Universal Robots URScript: camisa.script

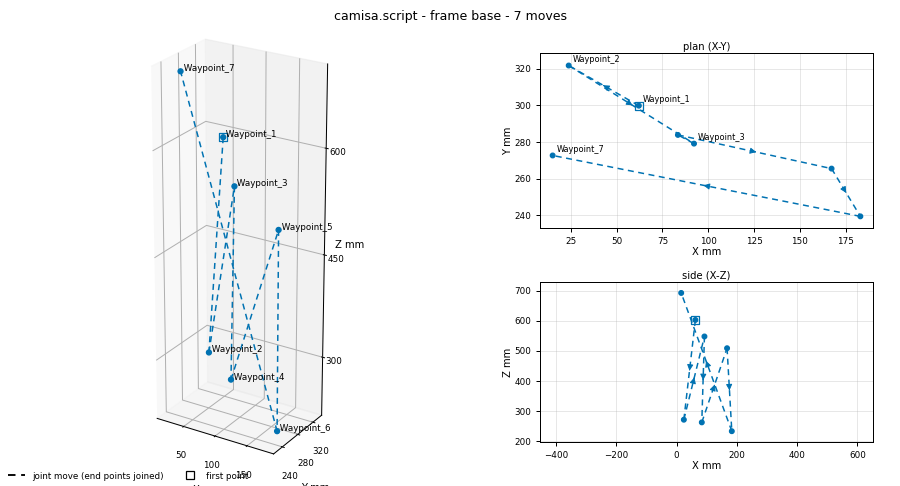
[picture p0: tool path of camisa.script in frame base, 7 of 7 moves have a stored position in this frame; points joined in program order, loops and branches not executed]
def camisa():
  set_tcp(p[0.0,0.0,0.0777,0.0,0.0,0.0])
  set_payload(0.1, [0.0, 0.0, 0.08])
  set_tool_voltage(24)
  set_gravity([0.0, 0.0, 9.82])
  modbus_add_signal("192.168.3.71", 255, 129, 3, "RX74", False)
  modbus_set_signal_update_frequency("RX74", 10)
  modbus_add_signal("192.168.3.133", 255, 130, 3, "TX71", False)
  modbus_set_signal_update_frequency("TX71", 10)
  modbus_set_runstate_dependent_choice("RX74",0)
  modbus_set_runstate_dependent_choice("TX71",0)
  set_standard_analog_input_domain(0, 1)
  set_standard_analog_input_domain(1, 1)
  set_tool_analog_input_domain(0, 1)
  set_tool_analog_input_domain(1, 1)
  set_analog_outputdomain(0, 0)
  set_analog_outputdomain(1, 0)
  set_input_actions_to_default()
  step_count_27ea16c7_09a7_48ac_b7d3_65c818ede42b = 0.0
  thread Step_Counter_Thread_a911c881_8547_437e_916d_f5c6adbcab51():
    while (True):
      step_count_27ea16c7_09a7_48ac_b7d3_65c818ede42b = step_count_27ea16c7_09a7_48ac_b7d3_65c818ede42b + 1.0
      sync()
    end
  end
  run Step_Counter_Thread_a911c881_8547_437e_916d_f5c6adbcab51()
  set_safety_mode_transition_hardness(1)
  global EVM=p[-0.15256820208455818,-0.42751336694884695,0.05022712170814066,-4.838863845671508E-5,-1.35928865028709E-4,-1.0092528187839596E-4]
  global EVM2=p[-0.29675101211797644,-0.4262716684008294,0.050741923201103156,4.332967508167418E-5,1.912443042895112E-4,1.5711081981983996E-4]
  global EVM3=p[0.0029371750612535727,-0.4263681938837632,0.05126173425663312,-1.739767729710799E-4,-4.4437664731219973E-5,-1.5069051907818709E-5]
  global FINAL=p[-0.22717262792356321,-0.43397417536669747,0.04266413451265917,1.4829527006895874E-4,-6.121065446531256E-5,-0.009247623504051445]
  global Plane_1=p[-0.3734029066127527,-0.3204511235418034,0.04435929145856908,9.783138506687844E-5,9.780306967539134E-5,-6.154211445520317E-5]
  global Plano4=p[-0.24996297948304783,-0.4275289861157397,0.05113872419679141,1.0348920676185259E-4,0.008007823293572955,-1.1342197607104979E-4]
  global cuervo_1=p[-0.3206063860027515,-0.4299262977046889,0.028915766646497074,-1.2221192979769074E-5,1.457304065347173E-4,-0.00918592635973644]
  global cuervo_2=p[-0.08949635923183384,-0.4299069312757706,0.028855734349918408,-2.0935967465238065E-4,-3.2568368129061994E-5,-1.9602101627311567E-4]
  global cuervo_3=p[0.1385881743231491,-0.4299379960100221,0.02888238485781129,-5.6603124500058476E-5,2.9018386427500325E-4,3.1643264082075785E-4]
  rtde_set_watchdog("speed_slider_mask", 10.0, "ignore")
  # begin: URCap Installation Node
  #   Source: OnRobot, 5.10.1, OnRobot A/S
  #   Type: Configuración de OnRobot
  # end: URCap Installation Node
  while (True):
    $ 1 "Robot Program"
    $ 2 "MoveJ"
    $ 3 "Waypoint_1" "breakAfter"
    movej(get_inverse_kin(p[.062136240038, .299828027685, .603022680044, -1.834983685346, -.149757239490, -.019890769577], qnear=[1.869443655014038, -1.4351256529437464, -0.7790663878070276, -1.2036622206317347, 1.3492110967636108, -0.03159171739687139]), a=1.3962634015954636, v=1.0471975511965976)
    $ 4 "Waypoint_2" "breakAfter"
    movej(get_inverse_kin(p[.023835907712, .321758372353, .271757076820, -1.863731925375, -.037561012054, .140144038975], qnear=[2.0221264362335205, -1.419579807912008, -2.544995371495382, 0.5165575742721558, 1.2549726963043213, 0.18266543745994568]), a=1.3962634015954636, v=1.0471975511965976)
    $ 5 "Waypoint_3" "breakAfter"
    movej(get_inverse_kin(p[.092250243875, .279124437920, .548122775729, -1.786373908672, -.042984052716, -.080491957922], qnear=[1.7929224967956543, -1.1799090544330042, -1.3519437948810022, -0.8312228361712855, 1.3243471384048462, -0.022686306630269826]), a=1.3962634015954636, v=1.0471975511965976)
    $ 6 "Waypoint_4" "breakAfter"
    movej(get_inverse_kin(p[.083456903249, .283883568854, .262945378806, -1.995978310655, -.014046129071, -.012538589481], qnear=[1.7989329099655151, -1.1812623182879847, -2.5902941862689417, 0.19511139392852783, 1.3615412712097168, 0.08338136970996857]), a=1.3962634015954636, v=1.0471975511965976)
    $ 7 "Waypoint_5" "breakAfter"
    movej(get_inverse_kin(p[.167347753731, .265482692449, .509106955622, -1.935792480015, .245397335100, -.242023934153], qnear=[1.4937984943389893, -1.2219527403460901, -1.3911832014666956, -0.9096539656268519, 1.356826663017273, 0.030969860032200813]), a=1.3962634015954636, v=1.0471975511965976)
    $ 8 "Waypoint_6" "breakAfter"
    movej(get_inverse_kin(p[.183070822697, .239415024508, .233639421906, -2.204298601929, .277917191407, -.134712347255], qnear=[1.27933931350708, -1.2732122580157679, -2.481180016194479, -0.03395682970155889, 1.6068198680877686, -0.019841496144429982]), a=1.3962634015954636, v=1.0471975511965976)
    $ 9 "Waypoint_7" "breakAfter"
    movej(get_inverse_kin(p[.015070981347, .272652259984, .692630508771, -1.570699931151, .003297320173, .159651201589], qnear=[3.173224687576294, -1.4638007322894495, -0.08294135728944951, -1.5549057165728968, 0.06875424832105637, 0.06481930613517761]), a=1.3962634015954636, v=1.0471975511965976)
  end
end
